(* CODESYS project Codesys_SAF_client.project

Project tree, tasks and I/O mapping:
  Device : CECC-LK, Festo AG & Co. KG, order no. 574418, version 3.5.7.27
    application Application
      libraries: Standard, * (System); CAA CiA 405, 3.5.7.0 (CAA Technical Workgroup); Solution Center Library, 3.5.8.0 (Festo Didactic SE - Customer Solution Center); CANbus, 3.5.7.0 (3S - Smart Software Solutions GmbH); Time and Date, 3.5.7.0 (3S - Smart Software Solutions GmbH); File Access, 3.5.7.0 (3S - Smart Software Solutions GmbH); Storage, 3.5.7.0 (3S - Smart Software Solutions GmbH); Util, * (System); CmpXMLParser, 3.5.5.0 (System)
      task MainTask (cyclic, interval t#20ms, priority 20) calls PLC_PRG
      program PLC_PRG [ST]
      global variables IO
    Onboard : CECC 14I/8O, Festo AG & Co. KG, version 3.4.5.5
        unmapped channels: Onboard Input, Onboard Output
      Digital Inputs
          unmapped channels: Onboard Input
      Digital Outputs
          unmapped channels: Onboard Output
    CAN : CANbus, 3S - Smart Software Solutions GmbH, version 3.5.10.0
        settings: Baudrate = 1000
      CANopen : CANopen_Manager, 3S - Smart Software Solutions GmbH, version 3.5.10.0
          settings: Sync CycleTime in Microseconds = 8000; Synchronous Window Length = 0; Enable Heartbeat generation = FALSE; Factory Settings Default = FALSE; Expert Settings Default = TRUE; ConfigVersion = 50659584
        BL20_GWBR_CANOPEN : BL20-GWBR-CANOPEN, TURCK, order no. 6827167, version Revision=16#00040017, FileVersion=4.23
            settings: General Options.Reset Node = FALSE; NODEIDSAVED = 2; SDO Timeout = 1000000; PDO_Autoconfig = TRUE; EXPERTSETTINGS = TRUE; Emergency-General Parameters.Emergency COBID = 16#00000082; Settings.COBID = 16#00000202; Settings.Transmission Type = 16#FF; Settings.available PDO-Parameter.Inhibit Time available = FALSE; Settings.available PDO-Parameter.Event Timer available = FALSE; Settings.Inhibit Time = 0; Settings.Event Timer = 0; Generic COBID = '$NODEID+16#0200'; Process by CANopenManager = TRUE; Settings.COBID = 16#00000302; Settings.Transmission Type = 16#FF; Settings.available PDO-Parameter.Inhibit Time available = FALSE; Settings.available PDO-Parameter.Event Timer available = FALSE; Settings.Inhibit Time = 0; Settings.Event Timer = 0; Generic COBID = '$NODEID+16#0300'; Process by CANopenManager = TRUE; Settings.COBID = 16#00000182; Settings.Transmission Type = 16#FF; Settings.available PDO-Parameter.Inhibit Time available = TRUE; Settings.available PDO-Parameter.Event Timer available = TRUE; Settings.Inhibit Time = 0; Settings.Event Timer = 0; Generic COBID = '$NODEID+16#0180'; Process by CANopenManager = TRUE; Settings.COBID = 16#00000282; Settings.Transmission Type = 16#FF; Settings.available PDO-Parameter.Inhibit Time available = TRUE; Settings.available PDO-Parameter.Event Timer available = TRUE; Settings.Inhibit Time = 0; Settings.Event Timer = 0; Generic COBID = '$NODEID+16#0280'; Process by CANopenManager = TRUE; WriteOutput8Bit : Generic_BL20_4DO.Index = 16#6200; WriteOutput8Bit : Generic_BL20_4DO.Subindex = 16#01;
              WriteOutput8Bit : Generic_BL20_4DO.ObjectLength = 8; WriteOutput8Bit : Generic_BL20_4DO_2.Index = 16#6200; WriteOutput8Bit : Generic_BL20_4DO_2.Subindex = 16#02; WriteOutput8Bit : Generic_BL20_4DO_2.ObjectLength = 4; WriteAnalogueOutput16 : Generic_BL20_2AO.Index = 16#6411; WriteAnalogueOutput16 : Generic_BL20_2AO.Subindex = 16#01; WriteAnalogueOutput16 : Generic_BL20_2AO.ObjectLength = 16; WriteAnalogueOutput16 : Generic_BL20_2AO.Index = 16#6411; WriteAnalogueOutput16 : Generic_BL20_2AO.Subindex = 16#02; WriteAnalogueOutput16 : Generic_BL20_2AO.ObjectLength = 16; ReadInput8Bit : Generic_BL20_4DI.Index = 16#6000; ReadInput8Bit : Generic_BL20_4DI.Subindex = 16#01; ReadInput8Bit : Generic_BL20_4DI.ObjectLength = 8; ReadAnalogueInput16Bit : Generic_BL20_4AI.Index = 16#6401; ReadAnalogueInput16Bit : Generic_BL20_4AI.Subindex = 16#01; ReadAnalogueInput16Bit : Generic_BL20_4AI.ObjectLength = 16; ReadAnalogueInput16Bit : Generic_BL20_4AI.Index = 16#6401; ReadAnalogueInput16Bit : Generic_BL20_4AI.Subindex = 16#02; ReadAnalogueInput16Bit : Generic_BL20_4AI.ObjectLength = 16; ReadAnalogueInput16Bit : Generic_BL20_4AI.Index = 16#6401; ReadAnalogueInput16Bit : Generic_BL20_4AI.Subindex = 16#03; ReadAnalogueInput16Bit : Generic_BL20_4AI.ObjectLength = 16; ReadAnalogueInput16Bit : Generic_BL20_4AI.Index = 16#6401; ReadAnalogueInput16Bit : Generic_BL20_4AI.Subindex = 16#04; ReadAnalogueInput16Bit : Generic_BL20_4AI.ObjectLength = 16; SDO List.Set Guardtime.Index = 16#100C; SDO List.Set Guardtime.Subindex = 16#00; SDO List.Set Guardtime.Value = 16#00000000; SDO List.Set Guardtime.Size = 16; SDO List.Set Guardtime.AbortIfError = FALSE; SDO List.Set Guardtime.JumpToLine = FALSE; SDO List.Set Guardtime.Line = 0; SDO List.Set Lifetime.Index = 16#100D; SDO List.Set Lifetime.Subindex = 16#00; SDO List.Set Lifetime.Value = 16#00000000; SDO List.Set Lifetime.Size = 8; SDO List.Set Lifetime.AbortIfError = FALSE; SDO List.Set Lifetime.JumpToLine = FALSE; SDO List.Set Lifetime.Line = 0; SDO List.Disable Emcy CobID.Index = 16#1014;
              SDO List.Disable Emcy CobID.Subindex = 16#00; SDO List.Disable Emcy CobID.Value = 16#80000082; SDO List.Disable Emcy CobID.Size = 32; SDO List.Disable Emcy CobID.AbortIfError = FALSE; SDO List.Disable Emcy CobID.JumpToLine = FALSE; SDO List.Disable Emcy CobID.Line = 0; SDO List.Set Emcy CobID.Index = 16#1014; SDO List.Set Emcy CobID.Subindex = 16#00; SDO List.Set Emcy CobID.Value = 16#00000082; SDO List.Set Emcy CobID.Size = 32; SDO List.Set Emcy CobID.AbortIfError = FALSE; SDO List.Set Emcy CobID.JumpToLine = FALSE; SDO List.Set Emcy CobID.Line = 0; SDO List.Set Heartbeat Consumer.Index = 16#1016; SDO List.Set Heartbeat Consumer.Subindex = 16#01; SDO List.Set Heartbeat Consumer.Value = 0; SDO List.Set Heartbeat Consumer.Size = 32; SDO List.Set Heartbeat Consumer.AbortIfError = FALSE; SDO List.Set Heartbeat Consumer.JumpToLine = FALSE; SDO List.Set Heartbeat Consumer.Line = 0; SDO List.Set Heartbeat Producer.Index = 16#1017; SDO List.Set Heartbeat Producer.Subindex = 16#00; SDO List.Set Heartbeat Producer.Value = 16#00000000; SDO List.Set Heartbeat Producer.Size = 16; SDO List.Set Heartbeat Producer.AbortIfError = FALSE; SDO List.Set Heartbeat Producer.JumpToLine = FALSE; SDO List.Set Heartbeat Producer.Line = 0; SDO List.Disable PDO.Index = 16#1400; SDO List.Disable PDO.Subindex = 16#01; SDO List.Disable PDO.Value = 16#80000202; SDO List.Disable PDO.Size = 32; SDO List.Disable PDO.AbortIfError = FALSE; SDO List.Disable PDO.JumpToLine = FALSE; SDO List.Disable PDO.Line = 0; SDO List.Set transmission type.Index = 16#1400; SDO List.Set transmission type.Subindex = 16#02; SDO List.Set transmission type.Value = 16#FF; SDO List.Set transmission type.Size = 8; SDO List.Set transmission type.AbortIfError = FALSE; SDO List.Set transmission type.JumpToLine = FALSE;
              SDO List.Set transmission type.Line = 0; SDO List.Clear pdo mapping.Index = 16#1600; SDO List.Clear pdo mapping.Subindex = 16#00; SDO List.Clear pdo mapping.Value = 16#0; SDO List.Clear pdo mapping.Size = 8; SDO List.Clear pdo mapping.AbortIfError = FALSE; SDO List.Clear pdo mapping.JumpToLine = FALSE; SDO List.Clear pdo mapping.Line = 0; SDO List.Set Mapping.Index = 16#1600; SDO List.Set Mapping.Subindex = 16#01; SDO List.Set Mapping.Value = 16#62000108; SDO List.Set Mapping.Size = 32; SDO List.Set Mapping.AbortIfError = FALSE; SDO List.Set Mapping.JumpToLine = FALSE; SDO List.Set Mapping.Line = 0; SDO List.Set Mapping.Index = 16#1600; SDO List.Set Mapping.Subindex = 16#02; SDO List.Set Mapping.Value = 16#62000204; SDO List.Set Mapping.Size = 32; SDO List.Set Mapping.AbortIfError = FALSE; SDO List.Set Mapping.JumpToLine = FALSE; SDO List.Set Mapping.Line = 0; SDO List.Set number of mappings.Index = 16#1600; SDO List.Set number of mappings.Subindex = 16#00; SDO List.Set number of mappings.Value = 16#02; SDO List.Set number of mappings.Size = 8; SDO List.Set number of mappings.AbortIfError = FALSE; SDO List.Set number of mappings.JumpToLine = FALSE; SDO List.Set number of mappings.Line = 0; SDO List.Set and enable COB-ID.Index = 16#1400; SDO List.Set and enable COB-ID.Subindex = 16#01; SDO List.Set and enable COB-ID.Value = 16#00000202; SDO List.Set and enable COB-ID.Size = 32; SDO List.Set and enable COB-ID.AbortIfError = FALSE; SDO List.Set and enable COB-ID.JumpToLine = FALSE; SDO List.Set and enable COB-ID.Line = 0; SDO List.Disable PDO.Index = 16#1401; SDO List.Disable PDO.Subindex = 16#01; SDO List.Disable PDO.Value = 16#80000302; SDO List.Disable PDO.Size = 32;
              SDO List.Disable PDO.AbortIfError = FALSE; SDO List.Disable PDO.JumpToLine = FALSE; SDO List.Disable PDO.Line = 0; SDO List.Set transmission type.Index = 16#1401; SDO List.Set transmission type.Subindex = 16#02; SDO List.Set transmission type.Value = 16#FF; SDO List.Set transmission type.Size = 8; SDO List.Set transmission type.AbortIfError = FALSE; SDO List.Set transmission type.JumpToLine = FALSE; SDO List.Set transmission type.Line = 0; SDO List.Clear pdo mapping.Index = 16#1601; SDO List.Clear pdo mapping.Subindex = 16#00; SDO List.Clear pdo mapping.Value = 16#0; SDO List.Clear pdo mapping.Size = 8; SDO List.Clear pdo mapping.AbortIfError = FALSE; SDO List.Clear pdo mapping.JumpToLine = FALSE; SDO List.Clear pdo mapping.Line = 0; SDO List.Set Mapping.Index = 16#1601; SDO List.Set Mapping.Subindex = 16#01; SDO List.Set Mapping.Value = 16#64110110; SDO List.Set Mapping.Size = 32; SDO List.Set Mapping.AbortIfError = FALSE; SDO List.Set Mapping.JumpToLine = FALSE; SDO List.Set Mapping.Line = 0; SDO List.Set Mapping.Index = 16#1601; SDO List.Set Mapping.Subindex = 16#02; SDO List.Set Mapping.Value = 16#64110210; SDO List.Set Mapping.Size = 32; SDO List.Set Mapping.AbortIfError = FALSE; SDO List.Set Mapping.JumpToLine = FALSE; SDO List.Set Mapping.Line = 0; SDO List.Set number of mappings.Index = 16#1601; SDO List.Set number of mappings.Subindex = 16#00; SDO List.Set number of mappings.Value = 16#02; SDO List.Set number of mappings.Size = 8; SDO List.Set number of mappings.AbortIfError = FALSE; SDO List.Set number of mappings.JumpToLine = FALSE; SDO List.Set number of mappings.Line = 0; SDO List.Set and enable COB-ID.Index = 16#1401; SDO List.Set and enable COB-ID.Subindex = 16#01;
              SDO List.Set and enable COB-ID.Value = 16#00000302; SDO List.Set and enable COB-ID.Size = 32; SDO List.Set and enable COB-ID.AbortIfError = FALSE; SDO List.Set and enable COB-ID.JumpToLine = FALSE; SDO List.Set and enable COB-ID.Line = 0; SDO List.Disable PDO.Index = 16#1800; SDO List.Disable PDO.Subindex = 16#01; SDO List.Disable PDO.Value = 16#80000182; SDO List.Disable PDO.Size = 32; SDO List.Disable PDO.AbortIfError = FALSE; SDO List.Disable PDO.JumpToLine = FALSE; SDO List.Disable PDO.Line = 0; SDO List.Set transmission type.Index = 16#1800; SDO List.Set transmission type.Subindex = 16#02; SDO List.Set transmission type.Value = 16#FF; SDO List.Set transmission type.Size = 8; SDO List.Set transmission type.AbortIfError = FALSE; SDO List.Set transmission type.JumpToLine = FALSE; SDO List.Set transmission type.Line = 0; SDO List.Set inhibit time.Index = 16#1800; SDO List.Set inhibit time.Subindex = 16#03; SDO List.Set inhibit time.Value = 16#0000; SDO List.Set inhibit time.Size = 16; SDO List.Set inhibit time.AbortIfError = FALSE; SDO List.Set inhibit time.JumpToLine = FALSE; SDO List.Set inhibit time.Line = 0; SDO List.Set event time.Index = 16#1800; SDO List.Set event time.Subindex = 16#05; SDO List.Set event time.Value = 16#0000; SDO List.Set event time.Size = 16; SDO List.Set event time.AbortIfError = FALSE; SDO List.Set event time.JumpToLine = FALSE; SDO List.Set event time.Line = 0; SDO List.Clear pdo mapping.Index = 16#1A00; SDO List.Clear pdo mapping.Subindex = 16#00; SDO List.Clear pdo mapping.Value = 16#0; SDO List.Clear pdo mapping.Size = 8; SDO List.Clear pdo mapping.AbortIfError = FALSE; SDO List.Clear pdo mapping.JumpToLine = FALSE; SDO List.Clear pdo mapping.Line = 0;
              SDO List.Set Mapping.Index = 16#1A00; SDO List.Set Mapping.Subindex = 16#01; SDO List.Set Mapping.Value = 16#60000108; SDO List.Set Mapping.Size = 32; SDO List.Set Mapping.AbortIfError = FALSE; SDO List.Set Mapping.JumpToLine = FALSE; SDO List.Set Mapping.Line = 0; SDO List.Set number of mappings.Index = 16#1A00; SDO List.Set number of mappings.Subindex = 16#00; SDO List.Set number of mappings.Value = 16#01; SDO List.Set number of mappings.Size = 8; SDO List.Set number of mappings.AbortIfError = FALSE; SDO List.Set number of mappings.JumpToLine = FALSE; SDO List.Set number of mappings.Line = 0; SDO List.Set and enable COB-ID.Index = 16#1800; SDO List.Set and enable COB-ID.Subindex = 16#01; SDO List.Set and enable COB-ID.Value = 16#00000182; SDO List.Set and enable COB-ID.Size = 32; SDO List.Set and enable COB-ID.AbortIfError = FALSE; SDO List.Set and enable COB-ID.JumpToLine = FALSE; SDO List.Set and enable COB-ID.Line = 0; SDO List.Disable PDO.Index = 16#1801; SDO List.Disable PDO.Subindex = 16#01; SDO List.Disable PDO.Value = 16#80000282; SDO List.Disable PDO.Size = 32; SDO List.Disable PDO.AbortIfError = FALSE; SDO List.Disable PDO.JumpToLine = FALSE; SDO List.Disable PDO.Line = 0; SDO List.Set transmission type.Index = 16#1801; SDO List.Set transmission type.Subindex = 16#02; SDO List.Set transmission type.Value = 16#FF; SDO List.Set transmission type.Size = 8; SDO List.Set transmission type.AbortIfError = FALSE; SDO List.Set transmission type.JumpToLine = FALSE; SDO List.Set transmission type.Line = 0; SDO List.Set inhibit time.Index = 16#1801; SDO List.Set inhibit time.Subindex = 16#03; SDO List.Set inhibit time.Value = 16#0000; SDO List.Set inhibit time.Size = 16; SDO List.Set inhibit time.AbortIfError = FALSE;
              SDO List.Set inhibit time.JumpToLine = FALSE; SDO List.Set inhibit time.Line = 0; SDO List.Set event time.Index = 16#1801; SDO List.Set event time.Subindex = 16#05; SDO List.Set event time.Value = 16#0000; SDO List.Set event time.Size = 16; SDO List.Set event time.AbortIfError = FALSE; SDO List.Set event time.JumpToLine = FALSE; SDO List.Set event time.Line = 0; SDO List.Clear pdo mapping.Index = 16#1A01; SDO List.Clear pdo mapping.Subindex = 16#00; SDO List.Clear pdo mapping.Value = 16#0; SDO List.Clear pdo mapping.Size = 8; SDO List.Clear pdo mapping.AbortIfError = FALSE; SDO List.Clear pdo mapping.JumpToLine = FALSE; SDO List.Clear pdo mapping.Line = 0; SDO List.Set Mapping.Index = 16#1A01; SDO List.Set Mapping.Subindex = 16#01; SDO List.Set Mapping.Value = 16#64010110; SDO List.Set Mapping.Size = 32; SDO List.Set Mapping.AbortIfError = FALSE; SDO List.Set Mapping.JumpToLine = FALSE; SDO List.Set Mapping.Line = 0; SDO List.Set Mapping.Index = 16#1A01; SDO List.Set Mapping.Subindex = 16#02; SDO List.Set Mapping.Value = 16#64010210; SDO List.Set Mapping.Size = 32; SDO List.Set Mapping.AbortIfError = FALSE; SDO List.Set Mapping.JumpToLine = FALSE; SDO List.Set Mapping.Line = 0; SDO List.Set Mapping.Index = 16#1A01; SDO List.Set Mapping.Subindex = 16#03; SDO List.Set Mapping.Value = 16#64010310; SDO List.Set Mapping.Size = 32; SDO List.Set Mapping.AbortIfError = FALSE; SDO List.Set Mapping.JumpToLine = FALSE; SDO List.Set Mapping.Line = 0; SDO List.Set Mapping.Index = 16#1A01; SDO List.Set Mapping.Subindex = 16#04; SDO List.Set Mapping.Value = 16#64010410;
              SDO List.Set Mapping.Size = 32; SDO List.Set Mapping.AbortIfError = FALSE; SDO List.Set Mapping.JumpToLine = FALSE; SDO List.Set Mapping.Line = 0; SDO List.Set number of mappings.Index = 16#1A01; SDO List.Set number of mappings.Subindex = 16#00; SDO List.Set number of mappings.Value = 16#04; SDO List.Set number of mappings.Size = 8; SDO List.Set number of mappings.AbortIfError = FALSE; SDO List.Set number of mappings.JumpToLine = FALSE; SDO List.Set number of mappings.Line = 0; SDO List.Set and enable COB-ID.Index = 16#1801; SDO List.Set and enable COB-ID.Subindex = 16#01; SDO List.Set and enable COB-ID.Value = 16#00000282; SDO List.Set and enable COB-ID.Size = 32; SDO List.Set and enable COB-ID.AbortIfError = FALSE; SDO List.Set and enable COB-ID.JumpToLine = FALSE; SDO List.Set and enable COB-ID.Line = 0; ConfigVersion = 50659584
          Generic_BL20_4DI : Generic BL20-4DI, TURCK, order no. 0, version Revision=16#00040017, FileVersion=4.23
              settings: Number of Params = 1; ReadInput8Bit : Generic_BL20_4DI.Index = 16#6000; ReadInput8Bit : Generic_BL20_4DI.Subindex = 16#01; ReadInput8Bit : Generic_BL20_4DI.Startbit = 0; ReadInput8Bit : Generic_BL20_4DI.Endbit = 3
              unmapped channels: ReadInput8Bit : Generic_BL20_4DI
          Generic_BL20_4DI_1 : Generic BL20-4DI, TURCK, order no. 0, version Revision=16#00040017, FileVersion=4.23
              settings: Number of Params = 1; ReadInput8Bit : Generic_BL20_4DI.Index = 16#6000; ReadInput8Bit : Generic_BL20_4DI.Subindex = 16#01; ReadInput8Bit : Generic_BL20_4DI.Startbit = 4; ReadInput8Bit : Generic_BL20_4DI.Endbit = 7
              unmapped channels: ReadInput8Bit : Generic_BL20_4DI
          Generic_BL20_BR_PF : Generic BL20-BR/-PF, TURCK, order no. 0, version Revision=16#00040017, FileVersion=4.23
          Generic_BL20_4DO : Generic BL20-4DO, TURCK, order no. 0, version Revision=16#00040017, FileVersion=4.23
              settings: Number of Params = 1; WriteOutput8Bit : Generic_BL20_4DO.Index = 16#6200; WriteOutput8Bit : Generic_BL20_4DO.Subindex = 16#01; WriteOutput8Bit : Generic_BL20_4DO.Startbit = 0; WriteOutput8Bit : Generic_BL20_4DO.Endbit = 3
              unmapped channels: WriteOutput8Bit : Generic_BL20_4DO
          Generic_BL20_4DO_1 : Generic BL20-4DO, TURCK, order no. 0, version Revision=16#00040017, FileVersion=4.23
              settings: Number of Params = 1; WriteOutput8Bit : Generic_BL20_4DO.Index = 16#6200; WriteOutput8Bit : Generic_BL20_4DO.Subindex = 16#01; WriteOutput8Bit : Generic_BL20_4DO.Startbit = 4; WriteOutput8Bit : Generic_BL20_4DO.Endbit = 7
              unmapped channels: WriteOutput8Bit : Generic_BL20_4DO
          Generic_BL20_4DO_2 : Generic BL20-4DO, TURCK, order no. 0, version Revision=16#00040017, FileVersion=4.23
              settings: Number of Params = 1; WriteOutput8Bit : Generic_BL20_4DO_2.Index = 16#6200; WriteOutput8Bit : Generic_BL20_4DO_2.Subindex = 16#02; WriteOutput8Bit : Generic_BL20_4DO_2.Startbit = 0; WriteOutput8Bit : Generic_BL20_4DO_2.Endbit = 3
              unmapped channels: WriteOutput8Bit : Generic_BL20_4DO_2
          Generic_BL20_4AI : Generic BL20-4AI, TURCK, order no. 0, version Revision=16#00040017, FileVersion=4.23
              settings: Number of Params = 4; ReadAnalogueInput16Bit : Generic_BL20_4AI.Index = 16#6401; ReadAnalogueInput16Bit : Generic_BL20_4AI.Subindex = 16#01; ReadAnalogueInput16Bit : Generic_BL20_4AI.Startbit = 0; ReadAnalogueInput16Bit : Generic_BL20_4AI.Endbit = 15; ReadAnalogueInput16Bit : Generic_BL20_4AI.Index = 16#6401; ReadAnalogueInput16Bit : Generic_BL20_4AI.Subindex = 16#02; ReadAnalogueInput16Bit : Generic_BL20_4AI.Startbit = 0; ReadAnalogueInput16Bit : Generic_BL20_4AI.Endbit = 15; ReadAnalogueInput16Bit : Generic_BL20_4AI.Index = 16#6401; ReadAnalogueInput16Bit : Generic_BL20_4AI.Subindex = 16#03; ReadAnalogueInput16Bit : Generic_BL20_4AI.Startbit = 0; ReadAnalogueInput16Bit : Generic_BL20_4AI.Endbit = 15; ReadAnalogueInput16Bit : Generic_BL20_4AI.Index = 16#6401; ReadAnalogueInput16Bit : Generic_BL20_4AI.Subindex = 16#04; ReadAnalogueInput16Bit : Generic_BL20_4AI.Startbit = 0; ReadAnalogueInput16Bit : Generic_BL20_4AI.Endbit = 15
              unmapped channels: ReadAnalogueInput16Bit : Generic_BL20_4AI, ReadAnalogueInput16Bit : Generic_BL20_4AI, ReadAnalogueInput16Bit : Generic_BL20_4AI, ReadAnalogueInput16Bit : Generic_BL20_4AI
          Generic_BL20_2AO : Generic BL20-2AO, TURCK, order no. 0, version Revision=16#00040017, FileVersion=4.23
              settings: Number of Params = 2; WriteAnalogueOutput16 : Generic_BL20_2AO.Index = 16#6411; WriteAnalogueOutput16 : Generic_BL20_2AO.Subindex = 16#01; WriteAnalogueOutput16 : Generic_BL20_2AO.Startbit = 0; WriteAnalogueOutput16 : Generic_BL20_2AO.Endbit = 15; WriteAnalogueOutput16 : Generic_BL20_2AO.Index = 16#6411; WriteAnalogueOutput16 : Generic_BL20_2AO.Subindex = 16#02; WriteAnalogueOutput16 : Generic_BL20_2AO.Startbit = 0; WriteAnalogueOutput16 : Generic_BL20_2AO.Endbit = 15
              unmapped channels: WriteAnalogueOutput16 : Generic_BL20_2AO, WriteAnalogueOutput16 : Generic_BL20_2AO
        DTM425 : DTM425, ifm electronic gmbh, order no. DTM425, version Revision=16#00000000, FileVersion=8.2, File=DTM425.eds
            settings: General Options.Reset Node = FALSE; NODEIDSAVED = 32; SDO Timeout = 1000000; PDO_Autoconfig = FALSE; EXPERTSETTINGS = TRUE; Emergency-General Parameters.Emergency COBID = 16#000000A0; PDO 16#1400.COBID = 16#00000220; Process by CANopenManager = TRUE; PDO 16#1401.COBID = 16#00000320; Process by CANopenManager = TRUE; PDO 16#1402.COBID = 16#00000420; Process by CANopenManager = TRUE; PDO 16#1403.COBID = 16#00000520; Process by CANopenManager = TRUE; PDO 16#1800.COBID = 16#000001A0; PDO 16#1800.Event Timer = 0; Process by CANopenManager = TRUE; PDO 16#1801.COBID = 16#000002A0; PDO 16#1801.Event Timer = 0; Process by CANopenManager = TRUE; PDO 16#1802.COBID = 16#000003A0; PDO 16#1802.Event Timer = 0; Process by CANopenManager = TRUE; PDO 16#1803.COBID = 16#000004A0; PDO 16#1803.Event Timer = 0; Process by CANopenManager = TRUE; Write Data (mappable): Write Trigger.Subindex = 16#00; Write Data (mappable): Data_sub1.Subindex = 16#01; Write Data (mappable): Data_sub2.Subindex = 16#02; Write Data (mappable): Data_sub3.Subindex = 16#03; Device Status.Subindex = 16#00; Read Data (mappable): Data_sub1.Subindex = 16#01; Read Data (mappable): Data_sub2.Subindex = 16#02; Read Data (mappable): Data_sub3.Subindex = 16#03; SDO List.Disable Emcy CobID.Index = 16#1014; SDO List.Disable Emcy CobID.Subindex = 16#00; SDO List.Disable Emcy CobID.Value = 16#800000A0; SDO List.Disable Emcy CobID.Size = 32; SDO List.Disable Emcy CobID.AbortIfError = FALSE; SDO List.Disable Emcy CobID.JumpToLine = FALSE;
              SDO List.Disable Emcy CobID.Line = 0; SDO List.Set Emcy CobID.Index = 16#1014; SDO List.Set Emcy CobID.Subindex = 16#00; SDO List.Set Emcy CobID.Value = 16#000000A0; SDO List.Set Emcy CobID.Size = 32; SDO List.Set Emcy CobID.AbortIfError = FALSE; SDO List.Set Emcy CobID.JumpToLine = FALSE; SDO List.Set Emcy CobID.Line = 0; SDO List.Set Heartbeat Producer.Index = 16#1017; SDO List.Set Heartbeat Producer.Subindex = 16#00; SDO List.Set Heartbeat Producer.Value = 16#00000000; SDO List.Set Heartbeat Producer.Size = 16; SDO List.Set Heartbeat Producer.AbortIfError = FALSE; SDO List.Set Heartbeat Producer.JumpToLine = FALSE; SDO List.Set Heartbeat Producer.Line = 0; SDO List.Disable PDO.Index = 16#1400; SDO List.Disable PDO.Subindex = 16#01; SDO List.Disable PDO.Value = 16#80000220; SDO List.Disable PDO.Size = 32; SDO List.Disable PDO.AbortIfError = FALSE; SDO List.Disable PDO.JumpToLine = FALSE; SDO List.Disable PDO.Line = 0; SDO List.Set transmission type.Index = 16#1400; SDO List.Set transmission type.Subindex = 16#02; SDO List.Set transmission type.Value = 16#FF; SDO List.Set transmission type.Size = 8; SDO List.Set transmission type.AbortIfError = FALSE; SDO List.Set transmission type.JumpToLine = FALSE; SDO List.Set transmission type.Line = 0; SDO List.Clear pdo mapping.Index = 16#1600; SDO List.Clear pdo mapping.Subindex = 16#00; SDO List.Clear pdo mapping.Value = 16#0; SDO List.Clear pdo mapping.Size = 8; SDO List.Clear pdo mapping.AbortIfError = FALSE; SDO List.Clear pdo mapping.JumpToLine = FALSE; SDO List.Clear pdo mapping.Line = 0; SDO List.Set Mapping.Index = 16#1600; SDO List.Set Mapping.Subindex = 16#01; SDO List.Set Mapping.Value = 16#230F0040; SDO List.Set Mapping.Size = 32;
              SDO List.Set Mapping.AbortIfError = FALSE; SDO List.Set Mapping.JumpToLine = FALSE; SDO List.Set Mapping.Line = 0; SDO List.Set number of mappings.Index = 16#1600; SDO List.Set number of mappings.Subindex = 16#00; SDO List.Set number of mappings.Value = 16#01; SDO List.Set number of mappings.Size = 8; SDO List.Set number of mappings.AbortIfError = FALSE; SDO List.Set number of mappings.JumpToLine = FALSE; SDO List.Set number of mappings.Line = 0; SDO List.Set and enable COB-ID.Index = 16#1400; SDO List.Set and enable COB-ID.Subindex = 16#01; SDO List.Set and enable COB-ID.Value = 16#00000220; SDO List.Set and enable COB-ID.Size = 32; SDO List.Set and enable COB-ID.AbortIfError = FALSE; SDO List.Set and enable COB-ID.JumpToLine = FALSE; SDO List.Set and enable COB-ID.Line = 0; SDO List.Disable PDO.Index = 16#1401; SDO List.Disable PDO.Subindex = 16#01; SDO List.Disable PDO.Value = 16#80000320; SDO List.Disable PDO.Size = 32; SDO List.Disable PDO.AbortIfError = FALSE; SDO List.Disable PDO.JumpToLine = FALSE; SDO List.Disable PDO.Line = 0; SDO List.Set transmission type.Index = 16#1401; SDO List.Set transmission type.Subindex = 16#02; SDO List.Set transmission type.Value = 16#FF; SDO List.Set transmission type.Size = 8; SDO List.Set transmission type.AbortIfError = FALSE; SDO List.Set transmission type.JumpToLine = FALSE; SDO List.Set transmission type.Line = 0; SDO List.Clear pdo mapping.Index = 16#1601; SDO List.Clear pdo mapping.Subindex = 16#00; SDO List.Clear pdo mapping.Value = 16#0; SDO List.Clear pdo mapping.Size = 8; SDO List.Clear pdo mapping.AbortIfError = FALSE; SDO List.Clear pdo mapping.JumpToLine = FALSE; SDO List.Clear pdo mapping.Line = 0; SDO List.Set Mapping.Index = 16#1601; SDO List.Set Mapping.Subindex = 16#01;
              SDO List.Set Mapping.Value = 16#230A0140; SDO List.Set Mapping.Size = 32; SDO List.Set Mapping.AbortIfError = FALSE; SDO List.Set Mapping.JumpToLine = FALSE; SDO List.Set Mapping.Line = 0; SDO List.Set number of mappings.Index = 16#1601; SDO List.Set number of mappings.Subindex = 16#00; SDO List.Set number of mappings.Value = 16#01; SDO List.Set number of mappings.Size = 8; SDO List.Set number of mappings.AbortIfError = FALSE; SDO List.Set number of mappings.JumpToLine = FALSE; SDO List.Set number of mappings.Line = 0; SDO List.Set and enable COB-ID.Index = 16#1401; SDO List.Set and enable COB-ID.Subindex = 16#01; SDO List.Set and enable COB-ID.Value = 16#00000320; SDO List.Set and enable COB-ID.Size = 32; SDO List.Set and enable COB-ID.AbortIfError = FALSE; SDO List.Set and enable COB-ID.JumpToLine = FALSE; SDO List.Set and enable COB-ID.Line = 0; SDO List.Disable PDO.Index = 16#1402; SDO List.Disable PDO.Subindex = 16#01; SDO List.Disable PDO.Value = 16#80000420; SDO List.Disable PDO.Size = 32; SDO List.Disable PDO.AbortIfError = FALSE; SDO List.Disable PDO.JumpToLine = FALSE; SDO List.Disable PDO.Line = 0; SDO List.Set transmission type.Index = 16#1402; SDO List.Set transmission type.Subindex = 16#02; SDO List.Set transmission type.Value = 16#FF; SDO List.Set transmission type.Size = 8; SDO List.Set transmission type.AbortIfError = FALSE; SDO List.Set transmission type.JumpToLine = FALSE; SDO List.Set transmission type.Line = 0; SDO List.Clear pdo mapping.Index = 16#1602; SDO List.Clear pdo mapping.Subindex = 16#00; SDO List.Clear pdo mapping.Value = 16#0; SDO List.Clear pdo mapping.Size = 8; SDO List.Clear pdo mapping.AbortIfError = FALSE; SDO List.Clear pdo mapping.JumpToLine = FALSE; SDO List.Clear pdo mapping.Line = 0;
              SDO List.Set Mapping.Index = 16#1602; SDO List.Set Mapping.Subindex = 16#01; SDO List.Set Mapping.Value = 16#230A0240; SDO List.Set Mapping.Size = 32; SDO List.Set Mapping.AbortIfError = FALSE; SDO List.Set Mapping.JumpToLine = FALSE; SDO List.Set Mapping.Line = 0; SDO List.Set number of mappings.Index = 16#1602; SDO List.Set number of mappings.Subindex = 16#00; SDO List.Set number of mappings.Value = 16#01; SDO List.Set number of mappings.Size = 8; SDO List.Set number of mappings.AbortIfError = FALSE; SDO List.Set number of mappings.JumpToLine = FALSE; SDO List.Set number of mappings.Line = 0; SDO List.Set and enable COB-ID.Index = 16#1402; SDO List.Set and enable COB-ID.Subindex = 16#01; SDO List.Set and enable COB-ID.Value = 16#00000420; SDO List.Set and enable COB-ID.Size = 32; SDO List.Set and enable COB-ID.AbortIfError = FALSE; SDO List.Set and enable COB-ID.JumpToLine = FALSE; SDO List.Set and enable COB-ID.Line = 0; SDO List.Disable PDO.Index = 16#1403; SDO List.Disable PDO.Subindex = 16#01; SDO List.Disable PDO.Value = 16#80000520; SDO List.Disable PDO.Size = 32; SDO List.Disable PDO.AbortIfError = FALSE; SDO List.Disable PDO.JumpToLine = FALSE; SDO List.Disable PDO.Line = 0; SDO List.Set transmission type.Index = 16#1403; SDO List.Set transmission type.Subindex = 16#02; SDO List.Set transmission type.Value = 16#FF; SDO List.Set transmission type.Size = 8; SDO List.Set transmission type.AbortIfError = FALSE; SDO List.Set transmission type.JumpToLine = FALSE; SDO List.Set transmission type.Line = 0; SDO List.Clear pdo mapping.Index = 16#1603; SDO List.Clear pdo mapping.Subindex = 16#00; SDO List.Clear pdo mapping.Value = 16#0; SDO List.Clear pdo mapping.Size = 8; SDO List.Clear pdo mapping.AbortIfError = FALSE;
              SDO List.Clear pdo mapping.JumpToLine = FALSE; SDO List.Clear pdo mapping.Line = 0; SDO List.Set Mapping.Index = 16#1603; SDO List.Set Mapping.Subindex = 16#01; SDO List.Set Mapping.Value = 16#230A0340; SDO List.Set Mapping.Size = 32; SDO List.Set Mapping.AbortIfError = FALSE; SDO List.Set Mapping.JumpToLine = FALSE; SDO List.Set Mapping.Line = 0; SDO List.Set number of mappings.Index = 16#1603; SDO List.Set number of mappings.Subindex = 16#00; SDO List.Set number of mappings.Value = 16#01; SDO List.Set number of mappings.Size = 8; SDO List.Set number of mappings.AbortIfError = FALSE; SDO List.Set number of mappings.JumpToLine = FALSE; SDO List.Set number of mappings.Line = 0; SDO List.Set and enable COB-ID.Index = 16#1403; SDO List.Set and enable COB-ID.Subindex = 16#01; SDO List.Set and enable COB-ID.Value = 16#00000520; SDO List.Set and enable COB-ID.Size = 32; SDO List.Set and enable COB-ID.AbortIfError = FALSE; SDO List.Set and enable COB-ID.JumpToLine = FALSE; SDO List.Set and enable COB-ID.Line = 0; SDO List.Disable PDO.Index = 16#1800; SDO List.Disable PDO.Subindex = 16#01; SDO List.Disable PDO.Value = 16#800001A0; SDO List.Disable PDO.Size = 32; SDO List.Disable PDO.AbortIfError = FALSE; SDO List.Disable PDO.JumpToLine = FALSE; SDO List.Disable PDO.Line = 0; SDO List.Set transmission type.Index = 16#1800; SDO List.Set transmission type.Subindex = 16#02; SDO List.Set transmission type.Value = 16#FF; SDO List.Set transmission type.Size = 8; SDO List.Set transmission type.AbortIfError = FALSE; SDO List.Set transmission type.JumpToLine = FALSE; SDO List.Set transmission type.Line = 0; SDO List.Set inhibit time.Index = 16#1800; SDO List.Set inhibit time.Subindex = 16#03; SDO List.Set inhibit time.Value = 16#00C8;
              SDO List.Set inhibit time.Size = 16; SDO List.Set inhibit time.AbortIfError = FALSE; SDO List.Set inhibit time.JumpToLine = FALSE; SDO List.Set inhibit time.Line = 0; SDO List.Clear pdo mapping.Index = 16#1A00; SDO List.Clear pdo mapping.Subindex = 16#00; SDO List.Clear pdo mapping.Value = 16#0; SDO List.Clear pdo mapping.Size = 8; SDO List.Clear pdo mapping.AbortIfError = FALSE; SDO List.Clear pdo mapping.JumpToLine = FALSE; SDO List.Clear pdo mapping.Line = 0; SDO List.Set Mapping.Index = 16#1A00; SDO List.Set Mapping.Subindex = 16#01; SDO List.Set Mapping.Value = 16#21500020; SDO List.Set Mapping.Size = 32; SDO List.Set Mapping.AbortIfError = FALSE; SDO List.Set Mapping.JumpToLine = FALSE; SDO List.Set Mapping.Line = 0; SDO List.Set number of mappings.Index = 16#1A00; SDO List.Set number of mappings.Subindex = 16#00; SDO List.Set number of mappings.Value = 16#01; SDO List.Set number of mappings.Size = 8; SDO List.Set number of mappings.AbortIfError = FALSE; SDO List.Set number of mappings.JumpToLine = FALSE; SDO List.Set number of mappings.Line = 0; SDO List.Set and enable COB-ID.Index = 16#1800; SDO List.Set and enable COB-ID.Subindex = 16#01; SDO List.Set and enable COB-ID.Value = 16#000001A0; SDO List.Set and enable COB-ID.Size = 32; SDO List.Set and enable COB-ID.AbortIfError = FALSE; SDO List.Set and enable COB-ID.JumpToLine = FALSE; SDO List.Set and enable COB-ID.Line = 0; SDO List.Disable PDO.Index = 16#1801; SDO List.Disable PDO.Subindex = 16#01; SDO List.Disable PDO.Value = 16#800002A0; SDO List.Disable PDO.Size = 32; SDO List.Disable PDO.AbortIfError = FALSE; SDO List.Disable PDO.JumpToLine = FALSE; SDO List.Disable PDO.Line = 0; SDO List.Set transmission type.Index = 16#1801;
              SDO List.Set transmission type.Subindex = 16#02; SDO List.Set transmission type.Value = 16#FF; SDO List.Set transmission type.Size = 8; SDO List.Set transmission type.AbortIfError = FALSE; SDO List.Set transmission type.JumpToLine = FALSE; SDO List.Set transmission type.Line = 0; SDO List.Set inhibit time.Index = 16#1801; SDO List.Set inhibit time.Subindex = 16#03; SDO List.Set inhibit time.Value = 16#00C8; SDO List.Set inhibit time.Size = 16; SDO List.Set inhibit time.AbortIfError = FALSE; SDO List.Set inhibit time.JumpToLine = FALSE; SDO List.Set inhibit time.Line = 0; SDO List.Clear pdo mapping.Index = 16#1A01; SDO List.Clear pdo mapping.Subindex = 16#00; SDO List.Clear pdo mapping.Value = 16#0; SDO List.Clear pdo mapping.Size = 8; SDO List.Clear pdo mapping.AbortIfError = FALSE; SDO List.Clear pdo mapping.JumpToLine = FALSE; SDO List.Clear pdo mapping.Line = 0; SDO List.Set Mapping.Index = 16#1A01; SDO List.Set Mapping.Subindex = 16#01; SDO List.Set Mapping.Value = 16#220A0140; SDO List.Set Mapping.Size = 32; SDO List.Set Mapping.AbortIfError = FALSE; SDO List.Set Mapping.JumpToLine = FALSE; SDO List.Set Mapping.Line = 0; SDO List.Set number of mappings.Index = 16#1A01; SDO List.Set number of mappings.Subindex = 16#00; SDO List.Set number of mappings.Value = 16#01; SDO List.Set number of mappings.Size = 8; SDO List.Set number of mappings.AbortIfError = FALSE; SDO List.Set number of mappings.JumpToLine = FALSE; SDO List.Set number of mappings.Line = 0; SDO List.Set and enable COB-ID.Index = 16#1801; SDO List.Set and enable COB-ID.Subindex = 16#01; SDO List.Set and enable COB-ID.Value = 16#000002A0; SDO List.Set and enable COB-ID.Size = 32; SDO List.Set and enable COB-ID.AbortIfError = FALSE; SDO List.Set and enable COB-ID.JumpToLine = FALSE;
              SDO List.Set and enable COB-ID.Line = 0; SDO List.Disable PDO.Index = 16#1802; SDO List.Disable PDO.Subindex = 16#01; SDO List.Disable PDO.Value = 16#800003A0; SDO List.Disable PDO.Size = 32; SDO List.Disable PDO.AbortIfError = FALSE; SDO List.Disable PDO.JumpToLine = FALSE; SDO List.Disable PDO.Line = 0; SDO List.Set transmission type.Index = 16#1802; SDO List.Set transmission type.Subindex = 16#02; SDO List.Set transmission type.Value = 16#FF; SDO List.Set transmission type.Size = 8; SDO List.Set transmission type.AbortIfError = FALSE; SDO List.Set transmission type.JumpToLine = FALSE; SDO List.Set transmission type.Line = 0; SDO List.Set inhibit time.Index = 16#1802; SDO List.Set inhibit time.Subindex = 16#03; SDO List.Set inhibit time.Value = 16#00C8; SDO List.Set inhibit time.Size = 16; SDO List.Set inhibit time.AbortIfError = FALSE; SDO List.Set inhibit time.JumpToLine = FALSE; SDO List.Set inhibit time.Line = 0; SDO List.Clear pdo mapping.Index = 16#1A02; SDO List.Clear pdo mapping.Subindex = 16#00; SDO List.Clear pdo mapping.Value = 16#0; SDO List.Clear pdo mapping.Size = 8; SDO List.Clear pdo mapping.AbortIfError = FALSE; SDO List.Clear pdo mapping.JumpToLine = FALSE; SDO List.Clear pdo mapping.Line = 0; SDO List.Set Mapping.Index = 16#1A02; SDO List.Set Mapping.Subindex = 16#01; SDO List.Set Mapping.Value = 16#220A0240; SDO List.Set Mapping.Size = 32; SDO List.Set Mapping.AbortIfError = FALSE; SDO List.Set Mapping.JumpToLine = FALSE; SDO List.Set Mapping.Line = 0; SDO List.Set number of mappings.Index = 16#1A02; SDO List.Set number of mappings.Subindex = 16#00; SDO List.Set number of mappings.Value = 16#01; SDO List.Set number of mappings.Size = 8;
              SDO List.Set number of mappings.AbortIfError = FALSE; SDO List.Set number of mappings.JumpToLine = FALSE; SDO List.Set number of mappings.Line = 0; SDO List.Set and enable COB-ID.Index = 16#1802; SDO List.Set and enable COB-ID.Subindex = 16#01; SDO List.Set and enable COB-ID.Value = 16#000003A0; SDO List.Set and enable COB-ID.Size = 32; SDO List.Set and enable COB-ID.AbortIfError = FALSE; SDO List.Set and enable COB-ID.JumpToLine = FALSE; SDO List.Set and enable COB-ID.Line = 0; SDO List.Disable PDO.Index = 16#1803; SDO List.Disable PDO.Subindex = 16#01; SDO List.Disable PDO.Value = 16#800004A0; SDO List.Disable PDO.Size = 32; SDO List.Disable PDO.AbortIfError = FALSE; SDO List.Disable PDO.JumpToLine = FALSE; SDO List.Disable PDO.Line = 0; SDO List.Set transmission type.Index = 16#1803; SDO List.Set transmission type.Subindex = 16#02; SDO List.Set transmission type.Value = 16#FF; SDO List.Set transmission type.Size = 8; SDO List.Set transmission type.AbortIfError = FALSE; SDO List.Set transmission type.JumpToLine = FALSE; SDO List.Set transmission type.Line = 0; SDO List.Set inhibit time.Index = 16#1803; SDO List.Set inhibit time.Subindex = 16#03; SDO List.Set inhibit time.Value = 16#00C8; SDO List.Set inhibit time.Size = 16; SDO List.Set inhibit time.AbortIfError = FALSE; SDO List.Set inhibit time.JumpToLine = FALSE; SDO List.Set inhibit time.Line = 0; SDO List.Clear pdo mapping.Index = 16#1A03; SDO List.Clear pdo mapping.Subindex = 16#00; SDO List.Clear pdo mapping.Value = 16#0; SDO List.Clear pdo mapping.Size = 8; SDO List.Clear pdo mapping.AbortIfError = FALSE; SDO List.Clear pdo mapping.JumpToLine = FALSE; SDO List.Clear pdo mapping.Line = 0; SDO List.Set Mapping.Index = 16#1A03; SDO List.Set Mapping.Subindex = 16#01;
              SDO List.Set Mapping.Value = 16#220A0340; SDO List.Set Mapping.Size = 32; SDO List.Set Mapping.AbortIfError = FALSE; SDO List.Set Mapping.JumpToLine = FALSE; SDO List.Set Mapping.Line = 0; SDO List.Set number of mappings.Index = 16#1A03; SDO List.Set number of mappings.Subindex = 16#00; SDO List.Set number of mappings.Value = 16#01; SDO List.Set number of mappings.Size = 8; SDO List.Set number of mappings.AbortIfError = FALSE; SDO List.Set number of mappings.JumpToLine = FALSE; SDO List.Set number of mappings.Line = 0; SDO List.Set and enable COB-ID.Index = 16#1803; SDO List.Set and enable COB-ID.Subindex = 16#01; SDO List.Set and enable COB-ID.Value = 16#000004A0; SDO List.Set and enable COB-ID.Size = 32; SDO List.Set and enable COB-ID.AbortIfError = FALSE; SDO List.Set and enable COB-ID.JumpToLine = FALSE; SDO List.Set and enable COB-ID.Line = 0; ConfigVersion = 50659584
            unmapped channels: Write Data (mappable): Write Trigger, Write Data (mappable): Data_sub1, Write Data (mappable): Data_sub2, Write Data (mappable): Data_sub3, Device Status, Read Data (mappable): Data_sub1, Read Data (mappable): Data_sub2, Read Data (mappable): Data_sub3
*)

// Device/Application/IO
{attribute 'qualified_only'}
VAR_GLOBAL
		///////////////////////////
	// Inputs
	///////////////////////////
	
	xBG20		AT %IX1.0	: BOOL;	// Stopper released
	xBG21		AT %IX1.1	: BOOL;	// Carrier available
	xBG22		AT %IX1.2	: BOOL;	// Carrier ID bit 0
	xBG23		AT %IX1.3	: BOOL;	// Carrier ID bit 1
	xBG24		AT %IX1.4	: BOOL;	// Carrier ID bit 2
	xEmg		AT %IX0.0	: BOOL;	// Emergency stop
	
	///////////////////////////
	// Outputs
	///////////////////////////	
	
	xMB20		AT %QX1.0	: BOOL;	// Release stopper
	xQA1_LEFT	AT %QX0.5	: BOOL;	// Conveyor to the left
	xQA1_RIGHT	AT %QX0.4	: BOOL;	// Conveyor to the right
	xQA1_SLOW	AT %QX0.6	: BOOL;	// Conveyor Slow
	xQA1_STOP	AT %QX0.7	: BOOL;	// Conveyor Stop
	
END_VAR

// Device/Application/PLC_PRG
PROGRAM PLC_PRG
VAR

	State: UINT := 0;
	RFID: dc_ecp.Dtm425;
	RFID_DATA: dc_ecp.st_CPF_RfidData;
	Timer: TON;
	TCPclient: dc_ecp.TcpClientByteStream;
	corrcet_id: UINT;
	dataIn: STRING;
	dataOut: DWORD;
	date_and_time_var: DATE_AND_TIME;
	dateTimeOb: DTU.GetDateAndTime;
	xmlOb: DTU.GetDateAndTime;
	xml_end: EVTPARAM_CmpXMLEnd;
	xml_start: EVTPARAM_CmpXMLStart;
	xml_string_data_out: EVTPARAM_CmpXMLData;
	xml_string: STRING(200);
	send_size: UINT;
	xml_header: STRING := '<?xml version="1.0" encoding="UTF-8"?><p pn="';
	
	date_time_string: STRING;
	station_id: INT := 9;
	wait_time: TIME;
	strop_xml: INT;
	start_xml: INT;
	time_int: INT;
END_VAR

//timer(PT:=T#10S);
TCP();
RFID();
timer();

CASE State OF
	0: //Initialization
	IO.xQA1_RIGHT := TRUE;
	IO.xMB20 := TRUE;
	RFID.ClearError();
	TCP.Connect(sIP:='172.20.66.5', uiPort:=22000);
	State := 1;
	
	1: //wait for RIFD to clear
	IF RFID.xReady THEN
		RFID.Connect(usiNodeID := 32, usiNetworkId := 0, usiChannel :=1);
		State := 2;
	END_IF
		
	2: //wait for carrier
	IF IO.xBG21 = TRUE THEN
		IO.xMB20 := FALSE;
		IO.xQA1_RIGHT := FALSE;
		State := 4;
	END_IF

	4: //Read the RFID data
	IF RFID.xReady THEN
		RFID.ReadTag(uiStartAddress := 0, uiDataLength := SIZEOF(rfidData), ADR(rfidData));
		State := 5;
	END_IF

	5:
	IF RFID.xReady THEN
		carrierID:=dc_ecp.SwapWORD(rfidData.uiCarrierID);
		State := 6;
	END_IF
	
	6: //wait for RFID read.
	IF RFID.xReady THEN
		XML1 := WSTRING_TO_STRING("<?xml version='1.0' encoding='UTF-8'?><sensorreading><reading><carrierID>");
		XML2 := UINT_TO_STRING(carrierID);
		XML3 := WSTRING_TO_STRING("</carrierID><stationID>");
		XML4 := UINT_TO_STRING(stationID);
		XML5 := WSTRING_TO_STRING("</stationID></reading></sensorreading>");
		IF carrierID > 9 THEN
			det := 2;
		ELSE
			det := 1;
		END_IF
		FINALXML2 := CONCAT(CONCAT(CONCAT(CONCAT(XML1,XML2),XML3),XML4), XML5);
		State := 7;
	END_IF		
	
	7: //Make sure carrier is at the stopper.
	IF IO.xBG21 = TRUE THEN
		State := 8;
	END_IF
	
	8: //Send XML string to server for processing.
	IF TCP.xConnected AND TCP.xReady THEN
		TCP.Send(pToSend:=ADR(FINALXML2), uiSizeToSend:=135+det);
		State := 14;
	END_IF
	
	
	14: //Receive processing time from server
	IF TCP.xReady THEN
		TCP.Receive(pTOReceive:=ADR(dataIn), uiSizeToReceive:=SIZEOF(dataIn));
		IF STRING_TO_TIME(dataIN) > T#100MS THEN
			State := 15;
		END_IF
	END_IF

	 
	15: // Activate the Timer here:
	timer(IN:=TRUE, PT:= STRING_TO_TIME(dataIN));
	state := 16;
	
	16: //Wait for timer:
	IF timer.Q THEN
		timer(IN:=FALSE);
		State := 17;
	END_IF
	
	17:
		IO.xQA1_RIGHT := TRUE;
		IO.xMB20 := TRUE;
		dataIN := WSTRING_TO_STRING("T#0ms");
		State := 0;
 
END_CASE

END_PROGRAM
